// SIMATIC S7-200 project (STEP 7-Micro/WIN), CPU 221 REL 01.10

SYMBOL_TABLE USER1
START            I0.0
STOPP            I0.1
SENSOR_EXIT      I0.2     // cam bien canh tay robot quay ve
TANG1            M0.0     // cánh tay robot
TANG2            M0.1     // bang tai 1
SENSOR_UPPER     I0.3
SENSOR_MIDDLE    I0.4
SENSOR_LOWER     I0.5
TANG3            M0.2     // hang nho
TANG4            M0.3     // hang lon
TANG5            M0.4     // bang tai 2
TANG6            M0.6     // can gat
SENSOR_LON       I0.6
SENSOR_NHI       I0.7
END_SYMBOL_TABLE

ORGANIZATION_BLOCK MAIN:OB1
TITLE=PROGRAM COMMENTS
BEGIN
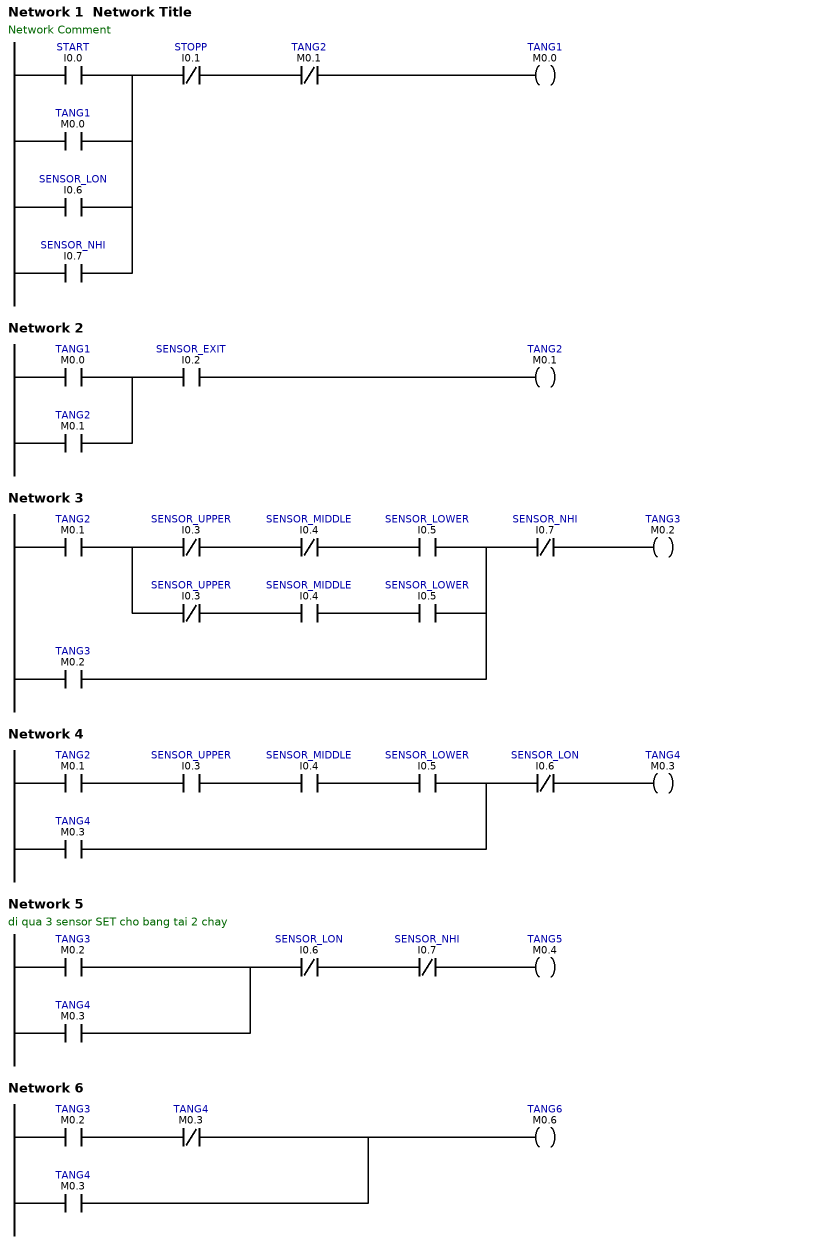
Network 1 // Network Title
// Network Comment
// (network saved uncompiled; LAD cells follow)
// row 0: c0 -| |- START:I0.0 v  c1 -|/|- STOPP:I0.1  c2 -|/|- TANG2:M0.1  c3 --  c4 -( ) TANG1:M0.0
// row 1: c0 -| |- TANG1:M0.0 ^v
// row 2: c0 -| |- SENSOR_LON:I0.6 ^v
// row 3: c0 -| |- SENSOR_NHI:I0.7 ^
Network 2
// (network saved uncompiled; LAD cells follow)
// row 0: c0 -| |- TANG1:M0.0 v  c1 -| |- SENSOR_EXIT:I0.2  c2 --  c3 --  c4 -( ) TANG2:M0.1
// row 1: c0 -| |- TANG2:M0.1 ^
Network 3
// (network saved uncompiled; LAD cells follow)
// row 0: c0 -| |- TANG2:M0.1 v  c1 -|/|- SENSOR_UPPER:I0.3  c2 -|/|- SENSOR_MIDDLE:I0.4  c3 -| |- SENSOR_LOWER:I0.5 v  c4 -|/|- SENSOR_NHI:I0.7  c5 -( ) TANG3:M0.2
// row 1: c0 ^  c1 -|/|- SENSOR_UPPER:I0.3  c2 -| |- SENSOR_MIDDLE:I0.4  c3 -| |- SENSOR_LOWER:I0.5 ^v
// row 2: c0 -| |- TANG3:M0.2  c1 --  c2 --  c3 -- ^
Network 4
// (network saved uncompiled; LAD cells follow)
// row 0: c0 -| |- TANG2:M0.1  c1 -| |- SENSOR_UPPER:I0.3  c2 -| |- SENSOR_MIDDLE:I0.4  c3 -| |- SENSOR_LOWER:I0.5 v  c4 -|/|- SENSOR_LON:I0.6  c5 -( ) TANG4:M0.3
// row 1: c0 -| |- TANG4:M0.3  c1 --  c2 --  c3 -- ^
Network 5
// di qua 3 sensor SET cho bang tai 2 chay
// (network saved uncompiled; LAD cells follow)
// row 0: c0 -| |- TANG3:M0.2  c1 -- v  c2 -|/|- SENSOR_LON:I0.6  c3 -|/|- SENSOR_NHI:I0.7  c4 -( ) TANG5:M0.4
// row 1: c0 -| |- TANG4:M0.3  c1 -- ^
Network 6
// (network saved uncompiled; LAD cells follow)
// row 0: c0 -| |- TANG3:M0.2  c1 -|/|- TANG4:M0.3  c2 -- v  c3 --  c4 -( ) TANG6:M0.6
// row 1: c0 -| |- TANG4:M0.3  c1 --  c2 -- ^
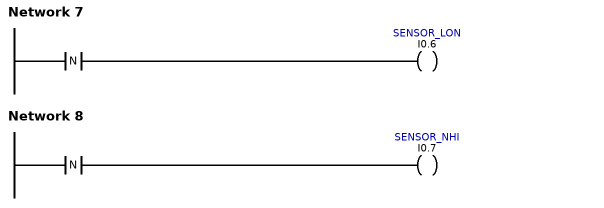
Network 7
// (network saved uncompiled; LAD cells follow)
// row 0: c0 -|N|-  c1 --  c2 --  c3 -( ) SENSOR_LON:I0.6
Network 8
// (network saved uncompiled; LAD cells follow)
// row 0: c0 -|N|-  c1 --  c2 --  c3 -( ) SENSOR_NHI:I0.7
END_ORGANIZATION_BLOCK
